% RSLogix 500 project I2P JOB 12_RUSSELL_BAK020.RSS, saved by version 10.00.00.00 %
PROJECT "ML02A"    % processor: Bul.1763 MicroLogix 1100 Series B %

PROGRAM FILES
  LAD 2   8 rungs

DATA FILES
  O0 OUTPUT  4 elements
  I1 INPUT  6 elements
  S2 STATUS  66 elements
  B3 BINARY  1 elements
  T4 TIMER  1 elements
  C5 COUNTER  1 elements
  R6 CONTROL  1 elements
  N7 INTEGER  1 elements
  F8 FLOAT  1 elements

LADDER 2
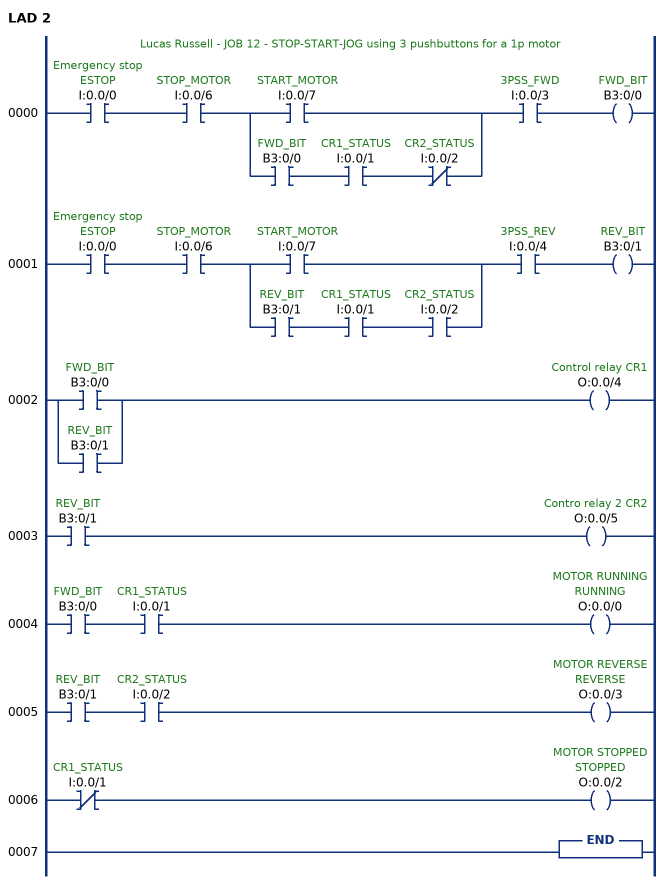
% Rung: 0 %
% Lucas Russell - JOB 12 - STOP-START-JOG using 3 pushbuttons for a 1p motor %
SOR XIC I:0.0/0 XIC I:0.0/6 BST XIC I:0.0/7 NXB XIC B3:0/0 XIC I:0.0/1 XIO I:0.0/2 BND XIC I:0.0/3 OTE B3:0/0 EOR
%   I:0.0/0  ESTOP  "Emergency stop" %
%   I:0.0/6  STOP_MOTOR %
%   I:0.0/7  START_MOTOR %
%   B3:0/0  "FWD_BIT" %
%   I:0.0/1  CR1_STATUS %
%   I:0.0/2  CR2_STATUS %
%   I:0.0/3  3PSS_FWD %
% Rung: 1 %
SOR XIC I:0.0/0 XIC I:0.0/6 BST XIC I:0.0/7 NXB XIC B3:0/1 XIC I:0.0/1 XIC I:0.0/2 BND XIC I:0.0/4 OTE B3:0/1 EOR
%   I:0.0/0  ESTOP  "Emergency stop" %
%   I:0.0/6  STOP_MOTOR %
%   I:0.0/7  START_MOTOR %
%   B3:0/1  "REV_BIT" %
%   I:0.0/1  CR1_STATUS %
%   I:0.0/2  CR2_STATUS %
%   I:0.0/4  3PSS_REV %
% Rung: 2 %
SOR BST XIC B3:0/0 NXB XIC B3:0/1 BND OTE O:0.0/4 EOR
%   B3:0/0  "FWD_BIT" %
%   B3:0/1  "REV_BIT" %
%   O:0.0/4  CR1  "Control relay" %
% Rung: 3 %
SOR XIC B3:0/1 OTE O:0.0/5 EOR
%   B3:0/1  "REV_BIT" %
%   O:0.0/5  CR2  "Contro relay 2" %
% Rung: 4 %
SOR XIC B3:0/0 XIC I:0.0/1 OTE O:0.0/0 EOR
%   B3:0/0  "FWD_BIT" %
%   I:0.0/1  CR1_STATUS %
%   O:0.0/0  RUNNING  "MOTOR RUNNING" %
% Rung: 5 %
SOR XIC B3:0/1 XIC I:0.0/2 OTE O:0.0/3 EOR
%   B3:0/1  "REV_BIT" %
%   I:0.0/2  CR2_STATUS %
%   O:0.0/3  REVERSE  "MOTOR REVERSE" %
% Rung: 6 %
SOR XIO I:0.0/1 OTE O:0.0/2 EOR
%   I:0.0/1  CR1_STATUS %
%   O:0.0/2  STOPPED  "MOTOR STOPPED" %
% Rung: 7 %
SOR END EOR

OTHER DOCUMENTED ADDRESSES
  B3:0/2  REV
  B3:1  FWD
  I:0.0/5  RUN_JOG  "Run/Jog Mode (A = Run, B - Jog)"
  I:0.0/8  JOG  "Normally open pushbutton"
  O:0.0/1  YELLOW_LIGHT  "Yellow light"
